// TIA Portal V17 export
// export: Created 2024-01-30T08:49:14.3599566Z, ExportSetting WithDefaults, DisplayName Totally Integrated Automation Portal, DisplayVersion V17 Update 6, DisplayName TIA Portal Openness, DisplayVersion V17 Update 6, DisplayName TIA Portal Version Control Interface, DisplayVersion V17, DisplayName STEP 7 Professional, DisplayVersion V17 Update 6, DisplayName STEP 7 Safety, DisplayVersion V17 Update 6, DisplayName WinCC Advanced, DisplayVersion V17 Update 6
DATA_BLOCK "PROGLOVE_TCP"   // DB32
{ S7_Optimized_Access := 'TRUE' }
VERSION : 0.1
// stored: AutoNumber true, DBAccessibleFromOPCUA true, DBAccessibleFromWebserver true, IsOnlyStoredInLoadMemory false, IsRetainMemResEnabled false, IsWriteProtectedInAS false, MemoryReserve 100
   VAR
      SEND_DATA { S7_SetPoint := 'True'} : String;
      RCV_DATA : String;
      TCON : Struct
         Done : Bool;
         Busy : Bool;
         Error : Bool;
         Status : Word;
      END_STRUCT;
   END_VAR
BEGIN
END_DATA_BLOCK
